PROGRAM pouS4Prompts
VAR
	


idbMsgPrompt: FB_CheckMessageBounds;
END_VAR

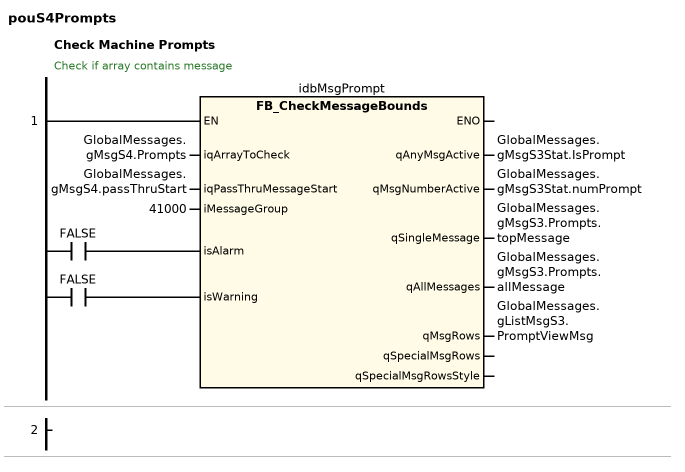
// NETWORK 1: Check Machine Prompts
// Check if array contains message
idbMsgPrompt(
    iqArrayToCheck := GlobalMessages.gMsgS4.Prompts,
    iqPassThruMessageStart := GlobalMessages.gMsgS4.passThruStart,
    iMessageGroup := 41000,
    isAlarm := FALSE,
    isWarning := FALSE,
    qAnyMsgActive => GlobalMessages.gMsgS3Stat.IsPrompt,
    qMsgNumberActive => GlobalMessages.gMsgS3Stat.numPrompt,
    qSingleMessage => GlobalMessages.gMsgS3.Prompts.topMessage,
    qAllMessages => GlobalMessages.gMsgS3.Prompts.allMessage,
    qMsgRows => GlobalMessages.gListMsgS3.PromptViewMsg); // FB_CheckMessageBounds

// NETWORK 2

END_PROGRAM

(* stored: Version 1.1.0.1, ProductVersion 3.1.4024.12
   POU pouS4Prompts: Id {da1db99f-f4b4-4307-97f8-6ec0cc41de57}, SpecialFunc None *)
